// TwinCAT 3 PLC project Untitled1
// ProgramVersion: 3.1.4024.0
// libraries:
//   Tc2_Standard, * (Beckhoff Automation GmbH)
//   Tc2_System, * (Beckhoff Automation GmbH)
//   Tc3_Module, * (Beckhoff Automation GmbH)
// project tree:
//   DUTs/ EnumType.TcDUT, StructType.TcDUT
//   / PlcTask.TcTTO
//   POUs/ MAIN.TcPOU
// real-time tasks:
//   TASK PlcTask: cycle T#10ms, priority 20, ADS port 350
// I/O:
//   DEVICE Device 1 (EtherCAT), AmsNetId 10.23.2.33.2.1
// variable links:
//   Untitled1 Instance <-> Device 1 (EtherCAT)
//     PlcTask Inputs/MAIN.myStructTypeVar.IO1 <-> Inputs/DevState

CONFIGURATION Untitled1
    RESOURCE PLC ON TwinCAT3
        TASK PlcTask(INTERVAL := T#10ms, PRIORITY := 20);
        PROGRAM MAIN WITH PlcTask : MAIN;
    END_RESOURCE
END_CONFIGURATION

// ---- DUTs/EnumType.TcDUT
{attribute 'qualified_only'}
{attribute 'strict'}
{attribute 'TO_STRING'}
TYPE EnumType :
(
	member1 := 0,
	member2,
	member3,
	member4
);
END_TYPE

// ---- DUTs/StructType.TcDUT
TYPE StructType :
STRUCT
	IO1 AT %I* : UINT;
	enumTypeVariable : EnumTYpe;
END_STRUCT
END_TYPE

// ---- POUs/MAIN.TcPOU
PROGRAM MAIN
VAR
	myStructTypeVar : StructType;
END_VAR

myStructTypeVar.enumTypeVariable := EnumType.member2;

END_PROGRAM
